// Mitsubishi GX Works2 project: Group15New   PLC: FX3G

// global labels: Global1
VAR_GLOBAL
  start_work_day AT X007 : BOOL;
  start_work_day_lamp AT Y007 : BOOL;
  cream_container AT D1100 : REAL;
  chocolate_container AT D1200 : REAL;
  biscuit_container AT D1300 : REAL;
  cream_amount AT D1400 : REAL;
  chocolate_amount AT D1500 : REAL;
  biscuit_amount AT D1600 : REAL;
  sprinkling_container AT D1700 : REAL;
  dipping_container AT D1800 : REAL;
END_VAR
VAR_GLOBAL CONSTANT
  const1 : REAL;
END_VAR
VAR_GLOBAL
  krembo_container AT D1900 : REAL;
  krembo_tray AT D2000 : REAL;
  end_work_day AT M20 : BOOL;
  lamp_blinking1 AT M30 : BOOL;
  lamp_blinking2 AT M40 : BOOL;
  lamp_finish_notice AT Y002 : BOOL;
END_VAR
VAR_GLOBAL CONSTANT
  cream_required : REAL := 300;
  biscuite_required : REAL := 6;
  chocolate_required_40 : REAL := 240;
END_VAR
VAR_GLOBAL
  cream_suitable_amount AT M50 : BOOL;
  biscuit_suitable_amount AT M60 : BOOL;
  chocolate_suitable_amount AT M70 : BOOL;
  TC_1 AT TC1 : BOOL;
  TS_1 AT TS1 : BOOL;
END_VAR
VAR_GLOBAL CONSTANT
  timer30 : INT := 30;
END_VAR
VAR_GLOBAL
  stop_blink_lamp AT M80 : BOOL;
  start_sprinkling AT X011 : BOOL;
  StartMachineA AT X010 : BOOL;
  MachineA_Stop AT X005 : BOOL;
  TouchSensor AT X003 : BOOL;
  TempSensorBelow15 AT X004 : BOOL;
  TempSensorAbove30 AT X002 : BOOL;
  Y_4 AT Y004 : BOOL;
  M_0 AT M90 : BOOL;
  MachineA_Status AT M100 : BOOL;
  camaraSensor AT X001 : BOOL;
  transport_A2B1 AT Y000 : BOOL;
  transport_A2B2 AT Y001 : BOOL;
  TC_2 AT TC2 : BOOL;
  TS_2 AT TS2 : BOOL;
  blink_continue AT M110 : BOOL;
  TS_3 AT TS3 : BOOL;
END_VAR
VAR_GLOBAL CONSTANT
  timer40 : INT := 40;
END_VAR
VAR_GLOBAL
  lamp_help AT M120 : BOOL;
END_VAR
VAR_GLOBAL CONSTANT
  sprrinkling_time : INT := 20;
END_VAR
VAR_GLOBAL
  end_sprinkling AT M130 : BOOL;
  TC_4 AT TC4 : BOOL;
  TS_4 AT TS4 : BOOL;
END_VAR
VAR_GLOBAL CONSTANT
  lamp_timer : INT := 10;
END_VAR
VAR_GLOBAL
  TC_5 AT TC5 : BOOL;
  TS_5 AT TS5 : BOOL;
  TC_3 AT TC3 : BOOL;
  transport_A2B AT M140 : BOOL;
  start_dipping AT X006 : BOOL;
  analog_input1 AT D8280 : INT;
  input_2_int AT D2010 : INT;
END_VAR
VAR_GLOBAL CONSTANT
  d_400 : INT := 390;
  const_5 : INT := 5;
  const_10 : INT := 10;
  chocolate_required_20 : REAL := 120;
END_VAR
VAR_GLOBAL
  analog_lamp AT M150 : BOOL;
  int_input AT D2020 : INT;
END_VAR
VAR_GLOBAL CONSTANT
  const_0 : INT;
END_VAR
VAR_GLOBAL
  TC_6 AT TC6 : BOOL;
  TS_6 AT TS6 : BOOL;
END_VAR
VAR_GLOBAL CONSTANT
  dipping_time : INT := 50;
END_VAR
VAR_GLOBAL
  dipping_lamp AT Y003 : BOOL;
  krembo_wrapping AT X000 : BOOL;
  CC_0 AT CC0 : BOOL;
  CS_0 AT CS0 : BOOL;
  CC_1 AT CC1 : BOOL;
  CS_1 AT CS1 : BOOL;
END_VAR
VAR_GLOBAL CONSTANT
  krembo_5 : INT := 5;
  krembo_6 : INT := 6;
END_VAR
VAR_GLOBAL
  analog_output AT D8282 : INT;
  total_krembo AT D2030 : REAL;
END_VAR
VAR_GLOBAL CONSTANT
  complete_tray : REAL := 6;
  mul_40 : REAL := 40;
END_VAR
VAR_GLOBAL
  TC_7 AT TC7 : BOOL;
  TS_7 AT TS7 : BOOL;
  TC_8 AT TC8 : BOOL;
  TS_8 AT TS8 : BOOL;
END_VAR
VAR_GLOBAL CONSTANT
  lamp_timer_day : INT := 5;
END_VAR

// task Task_01 (event TRUE, interval 0, priority 31): POU_01

PROGRAM POU_01
(* structured ladder/FBD written out as ST: instructions are called as NAME(EN, inputs, outputs); _pN, _eN, _tN stand for wires *)
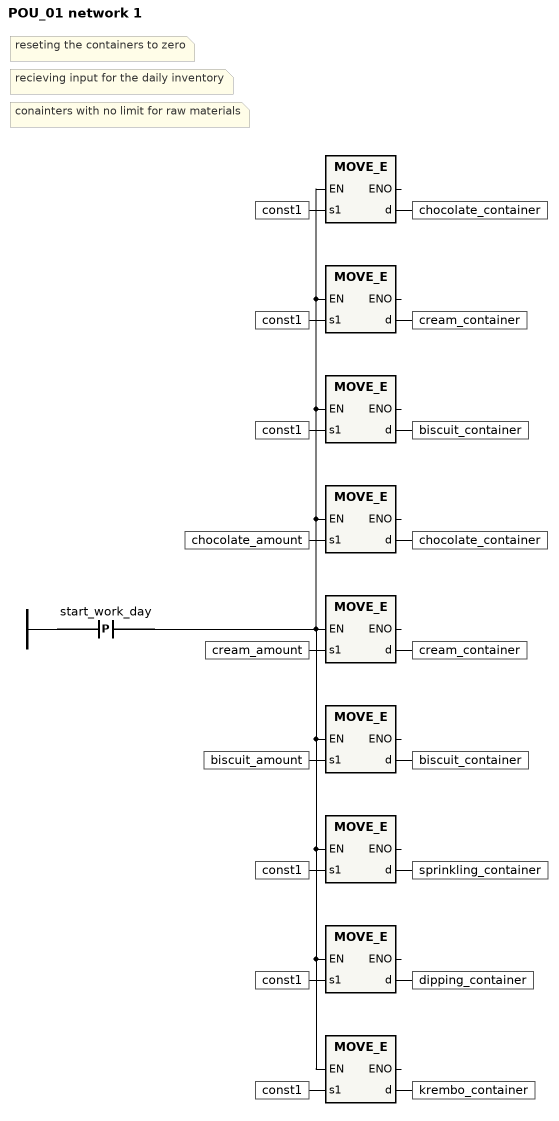
(* network 1 *)
(* reseting the containers to zero *)
(* recieving input for the daily inventory *)
(* conainters with no limit for raw materials *)
_p1 := LDP(TRUE, start_work_day);
MOVE_E(_p1, const1, chocolate_container);
MOVE_E(_p1, const1, cream_container);
MOVE_E(_p1, const1, biscuit_container);
MOVE_E(_p1, chocolate_amount, chocolate_container);
MOVE_E(_p1, cream_amount, cream_container);
MOVE_E(_p1, biscuit_amount, biscuit_container);
MOVE_E(_p1, const1, sprinkling_container);
MOVE_E(_p1, const1, dipping_container);
MOVE_E(_p1, const1, krembo_container);
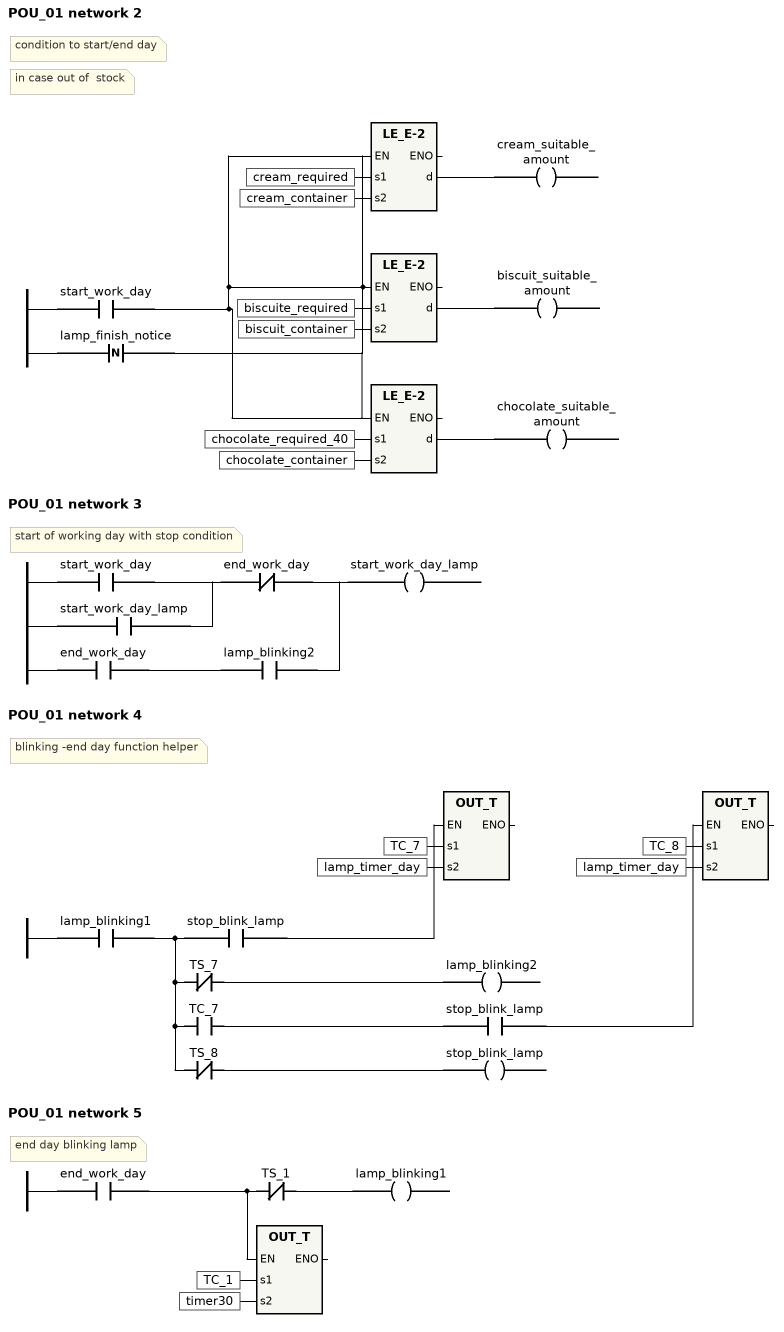
(* network 2 *)
(* condition to start/end day *)
(* in case out of  stock *)
_p1 := start_work_day OR LDF(TRUE, lamp_finish_notice);
LE_E(_p1, cream_required, cream_container, _t2);
cream_suitable_amount := _t2;
LE_E(_p1, biscuite_required, biscuit_container, _t3);
biscuit_suitable_amount := _t3;
LE_E(_p1, chocolate_required_40, chocolate_container, _t4);
chocolate_suitable_amount := _t4;
(* network 3 *)
(* start of working day with stop condition *)
start_work_day_lamp := ((start_work_day OR start_work_day_lamp) AND NOT end_work_day) OR (end_work_day AND lamp_blinking2);
(* network 4 *)
(* blinking -end day function helper *)
OUT_T(lamp_blinking1 AND stop_blink_lamp, TC_7, lamp_timer_day);
lamp_blinking2 := lamp_blinking1 AND NOT TS_7;
OUT_T(lamp_blinking1 AND TC_7 AND stop_blink_lamp, TC_8, lamp_timer_day);
stop_blink_lamp := lamp_blinking1 AND NOT TS_8;
(* network 5 *)
(* end day blinking lamp *)
lamp_blinking1 := end_work_day AND NOT TS_1;
OUT_T(end_work_day, TC_1, timer30);
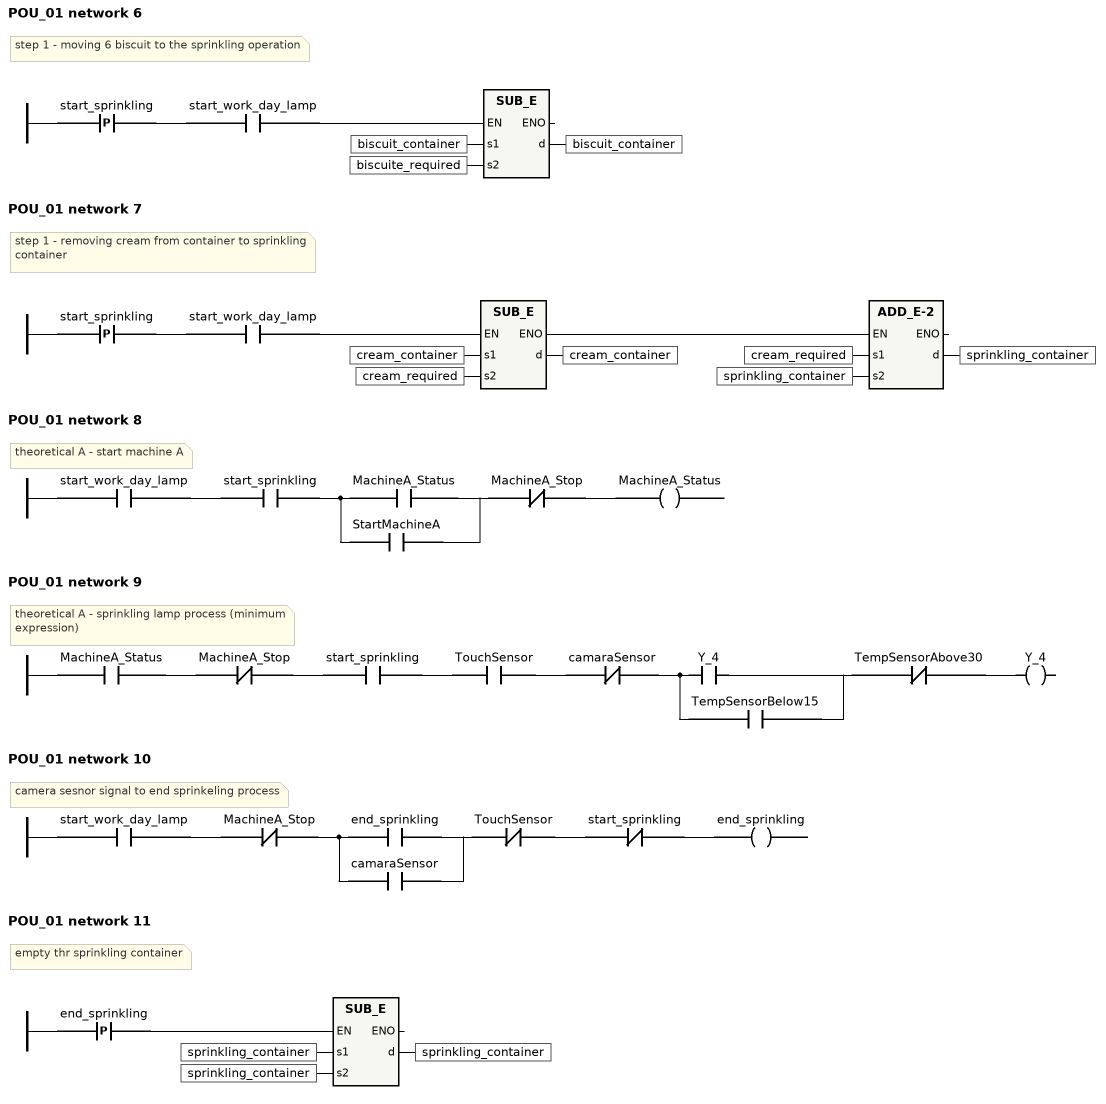
(* network 6 *)
(* step 1 - moving 6 biscuit to the sprinkling operation *)
SUB_E(LDP(TRUE, start_sprinkling) AND start_work_day_lamp, biscuit_container, biscuite_required, biscuit_container);
(* network 7 *)
(* step 1 - removing cream from container to sprinkling container *)
_e1 := SUB_E(LDP(TRUE, start_sprinkling) AND start_work_day_lamp, cream_container, cream_required, cream_container);
ADD_E(_e1, cream_required, sprinkling_container, sprinkling_container);
(* network 8 *)
(* theoretical A - start machine A *)
_p1 := start_work_day_lamp AND start_sprinkling;
MachineA_Status := ((_p1 AND MachineA_Status) OR (_p1 AND StartMachineA)) AND NOT MachineA_Stop;
(* network 9 *)
(* theoretical A - sprinkling lamp process (minimum expression) *)
_p1 := MachineA_Status AND NOT MachineA_Stop AND start_sprinkling AND TouchSensor AND NOT camaraSensor;
Y_4 := ((_p1 AND Y_4) OR (_p1 AND TempSensorBelow15)) AND NOT TempSensorAbove30;
(* network 10 *)
(* camera sesnor signal to end sprinkeling process *)
_p1 := start_work_day_lamp AND NOT MachineA_Stop;
end_sprinkling := (((_p1 AND end_sprinkling) OR (_p1 AND camaraSensor)) AND NOT TouchSensor) AND NOT start_sprinkling;
(* network 11 *)
(* empty thr sprinkling container *)
SUB_E(LDP(TRUE, end_sprinkling), sprinkling_container, sprinkling_container, sprinkling_container);
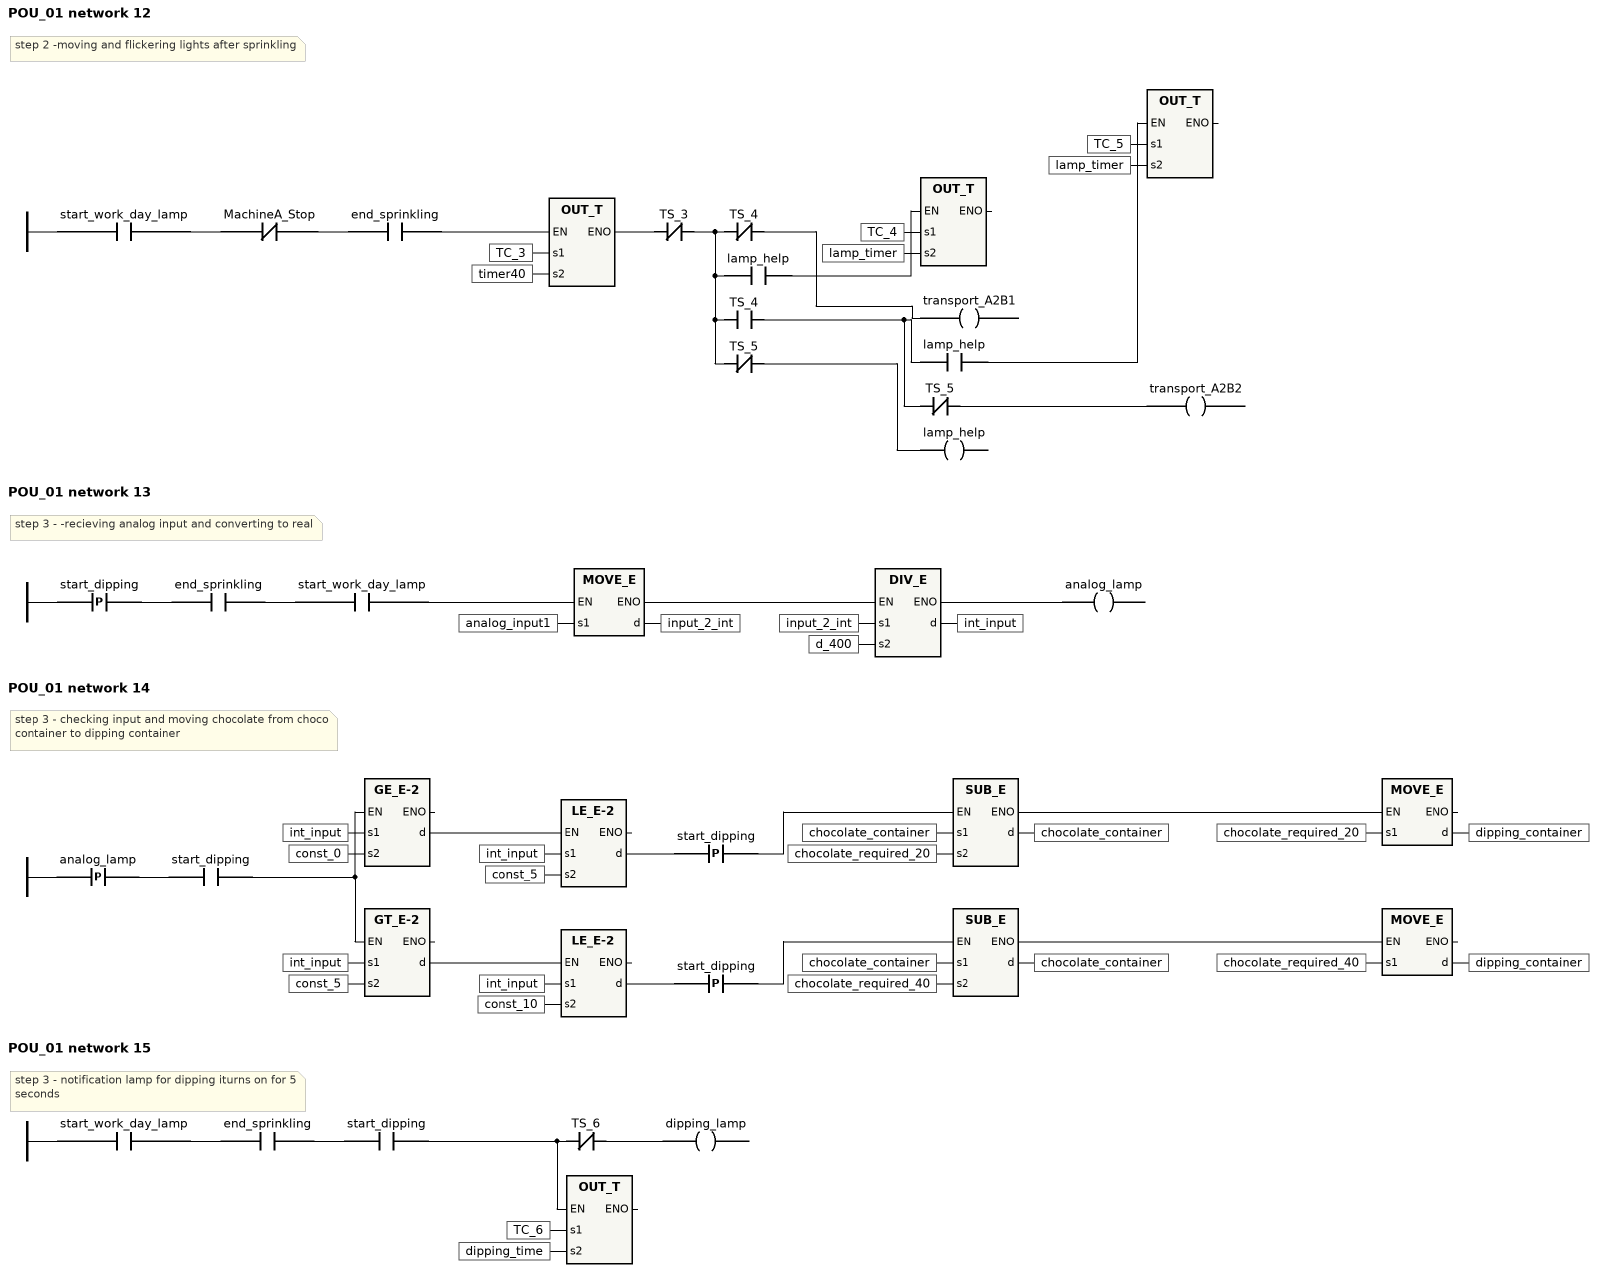
(* network 12 *)
(* step 2 -moving and flickering lights after sprinkling *)
_e1 := OUT_T(start_work_day_lamp AND NOT MachineA_Stop AND end_sprinkling, TC_3, timer40);
_p2 := _e1 AND NOT TS_3;
transport_A2B1 := _p2 AND NOT TS_4;
OUT_T(_p2 AND lamp_help, TC_4, lamp_timer);
_p3 := _p2 AND TS_4;
OUT_T(_p3 AND lamp_help, TC_5, lamp_timer);
transport_A2B2 := _p3 AND NOT TS_5;
lamp_help := _p2 AND NOT TS_5;
(* network 13 *)
(* step 3 - -recieving analog input and converting to real *)
_e1 := MOVE_E(LDP(TRUE, start_dipping) AND end_sprinkling AND start_work_day_lamp, analog_input1, input_2_int);
_e2 := DIV_E(_e1, input_2_int, d_400, int_input);
analog_lamp := _e2;
(* network 14 *)
(* step 3 - checking input and moving chocolate from choco container to dipping container *)
_p1 := LDP(TRUE, analog_lamp) AND start_dipping;
GE_E(_p1, int_input, const_0, _t2);
LE_E(_t2, int_input, const_5, _t3);
_e4 := SUB_E(_t3 AND LDP(TRUE, start_dipping), chocolate_container, chocolate_required_20, chocolate_container);
MOVE_E(_e4, chocolate_required_20, dipping_container);
GT_E(_p1, int_input, const_5, _t5);
LE_E(_t5, int_input, const_10, _t6);
_e7 := SUB_E(_t6 AND LDP(TRUE, start_dipping), chocolate_container, chocolate_required_40, chocolate_container);
MOVE_E(_e7, chocolate_required_40, dipping_container);
(* network 15 *)
(* step 3 - notification lamp for dipping iturns on for 5 seconds *)
_p1 := start_work_day_lamp AND end_sprinkling AND start_dipping;
dipping_lamp := _p1 AND NOT TS_6;
OUT_T(_p1, TC_6, dipping_time);
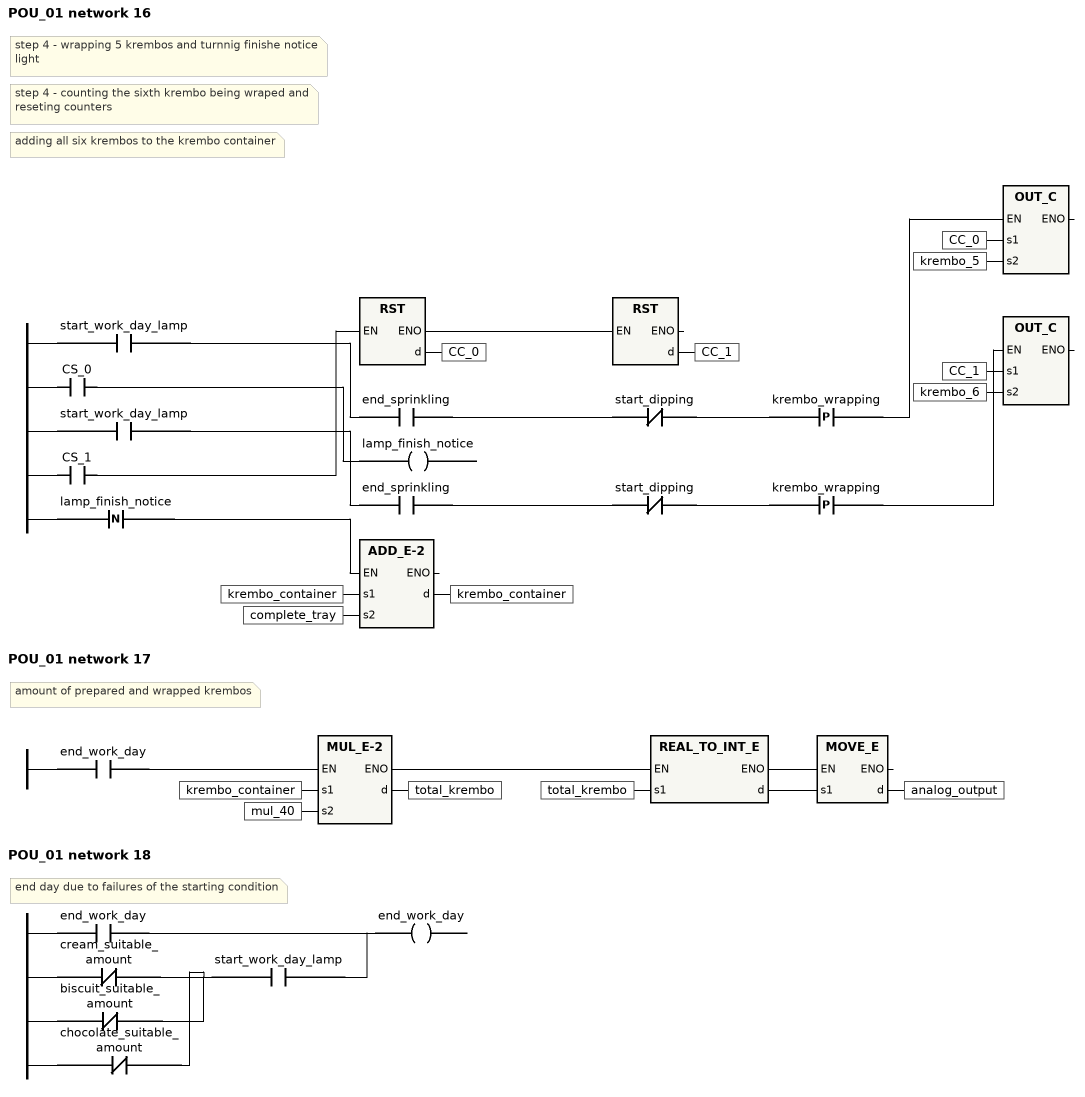
(* network 16 *)
(* step 4 - wrapping 5 krembos and turnnig finishe notice light *)
(* step 4 - counting the sixth krembo being wraped and reseting counters *)
(* adding all six krembos to the krembo container *)
OUT_C(start_work_day_lamp AND end_sprinkling AND NOT start_dipping AND LDP(TRUE, krembo_wrapping), CC_0, krembo_5);
lamp_finish_notice := CS_0;
OUT_C(start_work_day_lamp AND end_sprinkling AND NOT start_dipping AND LDP(TRUE, krembo_wrapping), CC_1, krembo_6);
_e1 := RST(CS_1, CC_0);
RST(_e1, CC_1);
ADD_E(LDF(TRUE, lamp_finish_notice), krembo_container, complete_tray, krembo_container);
(* network 17 *)
(* amount of prepared and wrapped krembos *)
_e1 := MUL_E(end_work_day, krembo_container, mul_40, total_krembo);
_e3 := REAL_TO_INT_E(_e1, total_krembo, _t2);
MOVE_E(_e3, _t2, analog_output);
(* network 18 *)
(* end day due to failures of the starting condition *)
end_work_day := end_work_day OR (((NOT cream_suitable_amount) OR (NOT biscuit_suitable_amount) OR (NOT chocolate_suitable_amount)) AND start_work_day_lamp);
END_PROGRAM
